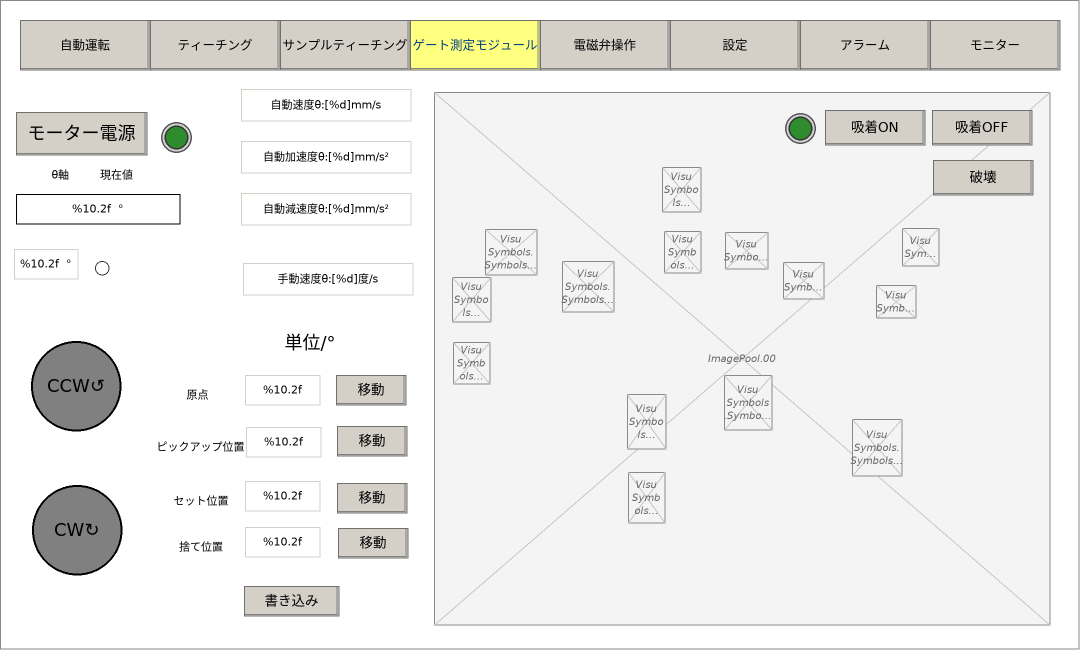
VISUALIZATION s_gm_teaching  // 1080x650
    Rectangle (0,0 1080x650)
    Image (434,92 616x533), image: ImagePool.00
    Label (35,160 51x30), "θ軸"
    Rectangle (16,194 164x30), "%10.2f °", text variable: gvl_axis.axisR.NcToPlc.ActPos
    Ellipse (31,341 90x90), "CCW↺"
        OnMouseDown: execute { gvl_visu.flg_btn_rotaryRigt := true; }
        OnMouseUp: execute { gvl_visu.flg_btn_rotaryRigt := FALSE; }
    Ellipse (32,485 90x90), "CW↻"
        OnMouseDown: execute { gvl_visu.flg_btn_rotaryLeft := TRUE; }
        OnMouseUp: execute { gvl_visu.flg_btn_rotaryLeft := FALSE; }
    Textfield (245,375 75x30), "%10.2f", text variable: gvl_visu.var_rotaryPos.origin
        OnMouseClick: write gvl_visu.var_rotaryPos.origin via VisuDialogs.Numpad
    Label (154,380 87x30), "原点"
    Textfield (246,427 75x30), "%10.2f", text variable: gvl_visu.var_rotaryPos.pickUp
        OnMouseClick: write gvl_visu.var_rotaryPos.pickUp via VisuDialogs.Numpad
    Label (159,432 83x30), "ピックアップ位置"
    Textfield (245,481 75x30), "%10.2f", text variable: gvl_visu.var_rotaryPos.set
        OnMouseClick: write gvl_visu.var_rotaryPos.set via VisuDialogs.Numpad
    Label (161,486 80x30), "セット位置"
    Lamp1 (159,120 35x35), variable: gvl_axis.fbi_mc_powerR.Busy, style: Lamp-Lamp1-Green
    Textfield (14,249 64x30), "%10.2f °", text variable: gvl_visu.var_gm_rotaryInch
        OnMouseClick: write gvl_visu.var_gm_rotaryInch via VisuDialogs.Numpad, format mm
    RadioButton (93,248 150x40), variable: gvl_visu.var_radio_rotaryJogMode
        Areas[0]: Text=インチ
        Areas[1]: Text=ジョグ
    Button (16,112 131x43), "モーター電源"
        toggle gvl_visu.flg_btn_gm_motorPower
    Button (244,586 95x30), "書き込み", colour toggle: gvl_visu.flg_btn_rotaryPos
        OnMouseClick: OpenDialog Dialog=d_gm_saveBtn, OpenModal=True, OpenCentered=True
    Button (336,375 70x30), "移動"
        tap gvl_visu.flg_btn_gm_moveOrigin
    Button (337,426 70x30), "移動"
        tap gvl_visu.flg_btn_gm_movePickUp
    Button (337,483 70x30), "移動"
        tap gvl_visu.flg_btn_gm_moveSet
    Textfield (241,89 170x32), "自動速度θ:[%d]mm/s", text variable: gvl_visu.var_gm_autoRotaryVel
        OnMouseClick: write gvl_visu.var_gm_autoRotaryVel via VisuDialogs.Numpad
    Textfield (241,141 170x32), "自動加速度θ:[%d]mm/s²", text variable: gvl_visu.var_gm_autoRotaryAcc
        OnMouseClick: write gvl_visu.var_gm_autoRotaryAcc via VisuDialogs.Numpad
    Textfield (241,193 170x32), "自動減速度θ:[%d]mm/s²", text variable: gvl_visu.var_gm_autoRotaryDec
        OnMouseClick: write gvl_visu.var_gm_autoRotaryDec via VisuDialogs.Numpad
    Button (20,20 130x50), "自動運転"
        OnMouseClick: change screen: s_auto
    Button (150,20 130x50), "ティーチング"
        OnMouseClick: change screen: s_teaching1
    Button (670,20 130x50), "設定"
        OnMouseClick: change screen: s_setting
    Button (540,20 130x50), "電磁弁操作"
        OnMouseClick: change screen: s_manual
    Button (410,20 130x50), "ゲート測定モジュール"
        OnMouseClick: change screen: s_gm_teaching
    Button (800,20 130x50), "アラーム", colour toggle: gvl_io.flg_signalTowerRed
        OnMouseClick: change screen: s_alarm
    Button (280,20 130x50), "サンプルティーチング"
        OnMouseClick: change screen: s_sample
    Label (252,328 116x30), "単位/°"
    Label (91,160 51x30), "現在値"
    Textfield (243,263 170x32), "手動速度θ:[%d]度/s", text variable: gvl_visu.var_gm_manualRotaryVel
        OnMouseClick: write gvl_visu.var_gm_manualRotaryVel via VisuDialogs.Numpad
    Textfield (245,527 75x30), "%10.2f", text variable: gvl_visu.var_rotaryPos.remove
        OnMouseClick: write gvl_visu.var_rotaryPos.remove via VisuDialogs.Numpad
    Label (161,532 80x30), "捨て位置"
    Button (338,528 70x30), "移動"
        tap gvl_visu.flg_btn_gm_moveRemove
    Image (562,261 52x51), angle 300, colour toggle: gvl_solv.ref_gm_rotary.in.in_flg_sensA, image: VisuSymbols.Symbols.ArrowQuarterLeftRight
        OnMouseDown: toggle gvl_visu.flg_btn_gm_svRotaryOrigin
    Image (485,229 52x46), angle 114, colour toggle: gvl_solv.ref_gm_rotary.in.in_flg_sensB, image: VisuSymbols.Symbols.ArrowQuarterRightLeft
        OnMouseDown: toggle gvl_visu.flg_btn_gm_svRotaryMoving
    Image (453,342 37x42), colour toggle: gvl_solv.ref_gm_pickUp.in.in_flg_sensA, image: VisuSymbols.Symbols.ArrowBoldDown
        OnMouseDown: toggle gvl_visu.flg_btn_gm_svPickUpOrigin
    Image (452,277 39x45), colour toggle: gvl_solv.ref_gm_pickUp.in.in_flg_sensB, image: VisuSymbols.Symbols.ArrowBoldUp
        OnMouseDown: toggle gvl_visu.flg_btn_gm_svPickUpMoving
    Image (876,285 40x33), angle 17, colour toggle: gvl_solv.ref_gm_chuck.in.in_flg_sensB, image: VisuSymbols.Symbols.ArrowBoldDown
        OnMouseDown: toggle gvl_visu.flg_btn_gm_svChuckClose
    Image (902,228 37x38), angle 17, colour toggle: gvl_solv.ref_gm_chuck.in.in_flg_sensA, image: VisuSymbols.Symbols.ArrowBoldUp
        OnMouseDown: toggle gvl_visu.flg_btn_gm_svChuckOpen
    Image (783,262 41x37), angle 299, colour toggle: gvl_solv.ref_gm_push.in.in_flg_sensB, image: VisuSymbols.Symbols.ArrowBoldLeftDown
        OnMouseDown: toggle gvl_visu.flg_btn_gm_svPushClose
    Image (725,232 43x37), angle 307, colour toggle: gvl_solv.ref_gm_push.in.in_flg_sensA, image: VisuSymbols.Symbols.ArrowBoldRightUp
        OnMouseDown: toggle gvl_visu.flg_btn_gm_svPushOpen
    Image (852,419 50x57), angle 290, colour toggle: gvl_solv.ref_gm_stamp.in.in_flg_sensB, image: VisuSymbols.Symbols.ArrowBoldDown
        OnMouseDown: toggle gvl_visu.flg_btn_gm_svStampMoving
    Image (724,375 48x55), angle 290, colour toggle: gvl_solv.ref_gm_stamp.in.in_flg_sensA, image: VisuSymbols.Symbols.ArrowBoldUp
        OnMouseDown: toggle gvl_visu.flg_btn_gm_svStampOrigin
    Image (627,394 39x55), colour toggle: gvl_elecylinder.ref_gm_axisTransport.input.in_flg_sensA, image: VisuSymbols.Symbols.ArrowBoldUp
        OnMouseDown: toggle gvl_visu.flg_btn_gm_eleTransportNegative
    Image (628,472 37x51), colour toggle: gvl_elecylinder.ref_gm_axisTransport.input.in_flg_sensB, image: VisuSymbols.Symbols.ArrowBoldDown
        OnMouseDown: toggle gvl_visu.flg_btn_gm_eleTransportPositive
    Image (662,167 39x45), colour toggle: gvl_elecylinder.ref_gm_axisPickUp.input.in_flg_sensA, image: VisuSymbols.Symbols.ArrowBoldUp
        OnMouseDown: toggle gvl_visu.flg_btn_gm_elePickUpNegative
    Image (664,231 37x42), colour toggle: gvl_elecylinder.ref_gm_axisPickUp.input.in_flg_sensB, image: VisuSymbols.Symbols.ArrowBoldDown
        OnMouseDown: toggle gvl_visu.flg_btn_gm_elePickUpPositive
    Button (825,110 100x35), "吸着ON"
        tap gvl_visu.flg_btn_gm_vacuumOn
    Button (933,160 100x35), "破壊"
        tap gvl_visu.flg_btn_gm_breakOn
    Button (932,110 100x35), "吸着OFF"
        tap gvl_visu.flg_btn_gm_vacuumOff
    Lamp1 (783,111 35x35), variable: gvl_solv.ref_gm_ejctor.input.in_flg_sensVac, style: Lamp-Lamp1-Green
    Button (930,20 130x50), "モニター"
        OnMouseClick: change screen: s_monitor
END_VISUALIZATION

(* stored: Version 1.1.0.1, ProductVersion 3.1.4024.11
   Visu s_gm_teaching: Id {7acaaefa-b222-436c-ac54-c20e624068da} *)
